(* Tx/Rx (string data) fifo control function block *)
FUNCTION_BLOCK FB_FrameFifo
VAR_INPUT
    bLog    : BOOL   := FALSE; (* TRUE => Enable log message output, FALSE => Disable *)
    sPrefix : STRING := 'Unknown::'; (* Log message description string (allows the identification of log message source) *)
    putObj  : STRING[25000];
    //	sPut		: T_MaxString 	:= ''; (* String message to add (write) to the fifo *)
END_VAR

VAR_OUTPUT
    bOk    : BOOL; (* TRUE = New entry added or removed succesfully, FALSE = Fifo overflow or fifo empty *)
    getObj : STRING[25000];
    nCount : UDINT := 0; (* Number of fifo entries *)
    cbFree : UDINT := 0; (* Free buffer space *)
END_VAR

VAR
    bReset                         : BOOL := TRUE;
    bAdd, bGet, bRelease, bGetFree : BOOL;
    cbSize                         : UDINT;
    fbBuffer                       : FB_MemRingBufferEx;
    buffer                         : ARRAY[-3..PLCPRJ_BUFFER_SIZE] OF BYTE; (* Internal buffer memory *)
    _Send                          : BOOL;
END_VAR

;

ACTION AddTail:
(* Adds new fifo entry *)
fbBuffer.A_AddTail(pBuffer  := ADR(buffer),
                   cbBuffer := SIZEOF(buffer),
                   pWrite   := ADR(putObj),
                   cbWrite  := SIZEOF(putObj),
                   bOk      => bOk,
                   nCount   => nCount,
                   cbSize   => cbSize,
                   cbFree   => cbFree);

IF bOk THEN
    cbFree := PLCPRJ_BUFFER_SIZE - fbBuffer.cbSize; (* Calculate the free buffer space *)

    IF bLog THEN (* Log message *)
        ADSLOGSTR(ADSLOG_MSGTYPE_HINT OR ADSLOG_MSGTYPE_LOG, CONCAT(sPrefix, '<="%s"'), putObj);
    END_IF
END_IF
END_ACTION

ACTION Clear:
(* Resets fifo = clears all data *)
fbBuffer.A_Reset(pBuffer  := ADR(buffer),
                 cbBuffer := SIZEOF(buffer),
                 bOk      => bOk,
                 nCount   => nCount,
                 cbSize   => cbSize,
                 cbFree   => cbFree);

cbFree := PLCPRJ_BUFFER_SIZE; (* Free buffer size *)
END_ACTION

ACTION RemoveHead:
(* Removes oldest fifo entry *)
fbBuffer.A_GetHead(pBuffer  := ADR(buffer),
                   cbBuffer := SIZEOF(buffer),
                   bOk      => bOk,
                   nCount   => nCount,
                   cbSize   => cbSize,
                   cbFree   => cbFree);

IF bOk THEN
    MEMCPY(ADR(getObj), fbBuffer.pRead, MIN(SIZEOF(getObj), fbBuffer.cbRead));
    cbFree := PLCPRJ_BUFFER_SIZE - fbBuffer.cbSize; (* Calculate the free buffer space *)

    fbBuffer.A_FreeHead(pBuffer  := ADR(buffer),
                        cbBuffer := SIZEOF(buffer),
                        bOk      => bOk,
                        nCount   => nCount,
                        cbSize   => cbSize,
                        cbFree   => cbFree);

    IF fbBuffer.bOk THEN
        ; (* Success *)
    ELSE
        ; (* Buffer empty *)
    END_IF
END_IF
END_ACTION

PROPERTY Send : BOOL
GET
Send := _Send;
END_GET
SET
_Send := Send;
END_SET
END_PROPERTY

END_FUNCTION_BLOCK

(* stored: Version 1.1.0.1
   POU FB_FrameFifo: Id {569e7401-3710-4598-aa05-b54586d01ffc}, SpecialFunc None
   Action AddTail: Id {9d0bf65e-4eae-4c60-aab3-4fa78b6cb7ba}
   Action Clear: Id {2d5c5598-7e6c-4d5d-a847-96a551240a71}
   Action RemoveHead: Id {09e2e3a4-2746-472b-aa8a-c0b08262dbf7}
   Property Send: Id {465b779d-cfd3-4a9d-a2a5-5ad1493f515f}
   Get Get: Id {6a4a3eb9-6046-4572-9f72-fc0eb3a5194f}
   Set Set: Id {99b805fd-bdf0-4058-a6c9-ef7c380e9cae} *)
